FUNCTION_BLOCK FB_PaperMachine
VAR_INPUT
	
	safetyCircuit		: BOOL;
	
END_VAR
VAR_OUTPUT
END_VAR
VAR
END_VAR


VAR_IN_OUT

	formingBoardSuctionRollDrive	: FB_DELTA_C2000_ETC;	
	formingBoardTractionRollDrive	: FB_DELTA_C2000_ETC;	

	stockPumpDrive	: FB_DELTA_C2000_ETC;	
	mixPumpDrive	: FB_DELTA_C2000_ETC;	
	wirePitPumpDrive	: FB_DELTA_C2000_ETC;	
	couchPitPumpDrive	: FB_DELTA_C2000_ETC;	

END_VAR

END_FUNCTION_BLOCK

(* stored: Version 1.1.0.1, ProductVersion 3.1.4024.15
   POU FB_PaperMachine: Id {4a8c14a2-6091-4cd1-afec-af3db8945cf3}, SpecialFunc None *)
